INTERFACE I_Base EXTENDS __SYSTEM.IQueryInterface

END_INTERFACE

(* stored: Version 1.1.0.1
   Itf I_Base: Id {6e8bc8ce-7f96-47dc-a8bc-48fb091ac6fd} *)
